FUNCTION_BLOCK Seq_Set_Plate_1 EXTENDS FB_Basis IMPLEMENTS I_Sequenz
VAR_INPUT
	// Skillzuweisung
	R_Move			:I_Skill_RoboterErweitert;
	G_Move			:I_Skill_SmartGreifer; 
	
	// Prozessparameter		
	RobParam				:ARRAY[0..4] OF sRoboterProzessVariablen;
	GripParam				:sSmartGreiferProzessVariablen;
	ErreichtParam			:ARRAY[0..1] OF sKraftVariablen;
END_VAR
VAR_OUTPUT
	
END_VAR
VAR
	
END_VAR

// Ablauf
ACT_Ablauf();

// Zustandshandling
CASE iState OF
	0:	// BEREIT
		IF bStart THEN
			bStart := FALSE;
			iState := 1;
		END_IF
	1:	// LAUFEND
		IF eSysCommand = 4 THEN
			bReset := TRUE;
			SFCReset := TRUE;
		END_IF
		
		IF bBeendet OR bReset THEN
			bReset := FALSE;
			SFCReset := FALSE;
			iState := 0;
		END_IF
END_CASE

ACTION ACT_Ablauf:
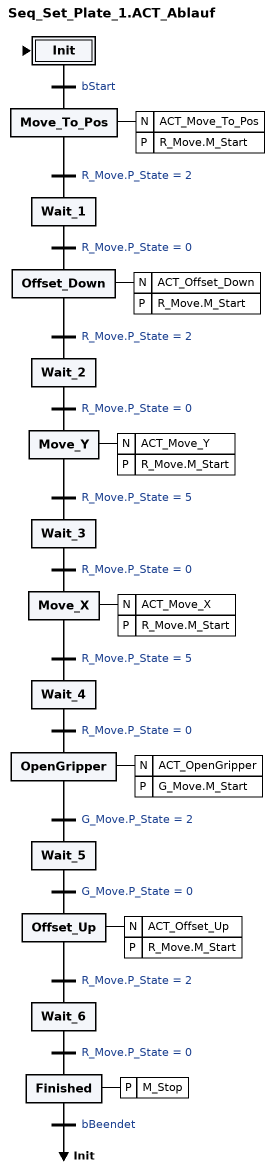
INITIAL_STEP Init:
END_STEP
TRANSITION FROM Init TO Move_To_Pos
    := bStart;
END_TRANSITION
STEP Move_To_Pos:
    ACT_Move_To_Pos(N);
    R_Move.M_Start(P);
END_STEP
TRANSITION FROM Move_To_Pos TO Wait_1
    := R_Move.P_State = 2;
END_TRANSITION
STEP Wait_1:
END_STEP
TRANSITION FROM Wait_1 TO Offset_Down
    := R_Move.P_State = 0;
END_TRANSITION
STEP Offset_Down:
    ACT_Offset_Down(N);
    R_Move.M_Start(P);
END_STEP
TRANSITION FROM Offset_Down TO Wait_2
    := R_Move.P_State = 2;
END_TRANSITION
STEP Wait_2:
END_STEP
TRANSITION FROM Wait_2 TO Move_Y
    := R_Move.P_State = 0;
END_TRANSITION
STEP Move_Y:
    ACT_Move_Y(N);
    R_Move.M_Start(P);
END_STEP
TRANSITION FROM Move_Y TO Wait_3
    := R_Move.P_State = 5;
END_TRANSITION
STEP Wait_3:
END_STEP
TRANSITION FROM Wait_3 TO Move_X
    := R_Move.P_State = 0;
END_TRANSITION
STEP Move_X:
    ACT_Move_X(N);
    R_Move.M_Start(P);
END_STEP
TRANSITION FROM Move_X TO Wait_4
    := R_Move.P_State = 5;
END_TRANSITION
STEP Wait_4:
END_STEP
TRANSITION FROM Wait_4 TO OpenGripper
    := R_Move.P_State = 0;
END_TRANSITION
STEP OpenGripper:
    ACT_OpenGripper(N);
    G_Move.M_Start(P);
END_STEP
TRANSITION FROM OpenGripper TO Wait_5
    := G_Move.P_State = 2;
END_TRANSITION
STEP Wait_5:
END_STEP
TRANSITION FROM Wait_5 TO Offset_Up
    := G_Move.P_State = 0;
END_TRANSITION
STEP Offset_Up:
    ACT_Offset_Up(N);
    R_Move.M_Start(P);
END_STEP
TRANSITION FROM Offset_Up TO Wait_6
    := R_Move.P_State = 2;
END_TRANSITION
STEP Wait_6:
END_STEP
TRANSITION FROM Wait_6 TO Finished
    := R_Move.P_State = 0;
END_TRANSITION
STEP Finished:
    M_Stop(P);
END_STEP
TRANSITION FROM Finished TO Init
    := bBeendet;
END_TRANSITION
END_ACTION

ACTION ACT_Move_To_Pos:
R_Move.P_RobotParam := RobParam[0];
END_ACTION

ACTION ACT_Move_X:
R_Move.P_RobotParam := RobParam[2];
R_Move.P_Erreicht := ErreichtParam[0];
END_ACTION

ACTION ACT_Move_Y:
R_Move.P_RobotParam := RobParam[3];
R_Move.P_Erreicht := ErreichtParam[1];
END_ACTION

ACTION ACT_Offset_Down:
R_Move.P_RobotParam := RobParam[1];
END_ACTION

ACTION ACT_Offset_Up:
R_Move.P_RobotParam := RobParam[4];
END_ACTION

ACTION ACT_OpenGripper:
G_Move.P_SGripperParam := GripParam;
END_ACTION

END_FUNCTION_BLOCK

(* stored: Version 1.1.0.1
   POU Seq_Set_Plate_1: Id {5bd25c77-6b1f-41ae-9003-3be438095eff}, SpecialFunc None
   Folder 01_Zuweisung: Id {56f46fb1-1341-4970-bd46-6b426e434d90}
   Action ACT_Ablauf: Id {ce1799b2-5359-4338-830f-378076096ef3}
   Action ACT_Move_To_Pos: Id {d405f6b9-7fa1-4db9-bcaf-3c7e78a02153}
   Action ACT_Move_X: Id {4f8366aa-2efb-46c3-93c2-f71cd50d16e5}
   Action ACT_Move_Y: Id {4c04199d-8fa5-4276-9d73-8d93d88b0f49}
   Action ACT_Offset_Down: Id {efad1f1d-2bcf-4788-8d80-abd10c9245e1}
   Action ACT_Offset_Up: Id {9aeb4cad-2868-4f66-8d70-66332615acea}
   Action ACT_OpenGripper: Id {15faffaf-20c3-495d-939b-545d9c8e7b08} *)
